FUNCTION_BLOCK FB_DataXMLP3_Old
VAR_INPUT
    	bSave:BOOL;
	    bRead:BOOL;

END_VAR
VAR_OUTPUT
    	bSaveParDone      :BOOL;
	    bReadParDone     :BOOL;
		bError                     :BOOL;		
END_VAR

VAR


	iDataSetp: INT;
	TON10:Tc2_Standard.TON;
	I1: INT;
	rt100:Tc2_Standard.R_TRIG;
	rt101:Tc2_Standard.R_TRIG;
	bExecute1: BOOL;
	bExecute2: BOOL;


	bSaveTemp: BOOL;
	bReadTemp: BOOL;

 fbXmlSrvWrite         : FB_XmlSrvWrite;
// fbXmlSrvWrite         : FB_SrvWrite;
   bExecuteW1             : BOOL;
   sFilePathPar_W       : T_MaxString ;

 
fbXmlSrvRead   : FB_XmlSrvRead;
//fbXmlSrvRead   : FB_SrvRead;
   bExecuteR          : BOOL;
   sFilePathPar_R      : T_MaxString ;
   sXPathR             : T_MaxString;
	AA: INT;
	BB: INT;












	handleTemp: UDINT;
END_VAR


M_WriteOrRead();

ACTION M_WriteOrRead:
bError := fbXmlSrvWrite.bError OR   fbXmlSrvRead.bError;

rt100(CLK:=bSave , Q=> );//保存参数
rt101(CLK:=bRead , Q=> );//读取参数

IF rt100.Q THEN  //保存参数
	iDataSetp:=100;
	TON10.IN:=FALSE;
	I1:=1;
	bExecute1:=FALSE;
	bExecute2:=FALSE;
	bSave:=FALSE;
	bRead:=FALSE;
    bSaveTemp:=TRUE;
	bReadTemp:=FALSE;
	bSaveParDone:=FALSE;
END_IF

IF rt101.Q THEN  //读取参数
	iDataSetp:=100;
	TON10.IN:=FALSE;
	I1:=1;
	bExecute1:=FALSE;
	bExecute2:=FALSE;	
	bSave:=FALSE;
	bRead:=FALSE;
    bReadTemp:=TRUE;
    bSaveTemp:=FALSE;
    bReadParDone:=FALSE;
END_IF

TON10(IN:= , PT:=T#200MS , Q=> , ET=> );

CASE  iDataSetp OF 
	
 100:
				CASE I1 OF 
				  1://轴参数
					sFilePathPar_W  := 'C:\P3XML\P3arrAxisParV2.xml';
					fbXmlSrvWrite.pSymAddr:=ADR(arrAxisParV2);
					fbXmlSrvWrite.cbSymSize:=SIZEOF(arrAxisParV2);   

					sFilePathPar_R  :=  'C:\P3XML\P3arrAxisParV2.xml';
					fbXmlSrvRead.pSymAddr:=ADR(arrAxisParV2);
					fbXmlSrvRead.cbSymSize:=SIZEOF(arrAxisParV2);   
     
				  2://arrTempPar
		  		    sFilePathPar_W  := 'C:\P3XML\P3arrTempPar.xml';
					fbXmlSrvWrite.pSymAddr:=ADR(arrTempPar);
					fbXmlSrvWrite.cbSymSize:=SIZEOF(arrTempPar);     

					sFilePathPar_R  := 'C:\P3XML\P3arrTempPar.xml';
					fbXmlSrvRead.pSymAddr:=ADR(arrTempPar);
					fbXmlSrvRead.cbSymSize:=SIZEOF(arrTempPar);   

				  3://P3par
		  		     sFilePathPar_W  := 'C:\P3XML\P3par.xml';
					fbXmlSrvWrite.pSymAddr:=ADR(P3par);
					fbXmlSrvWrite.cbSymSize:=SIZEOF(P3par);     

					sFilePathPar_R  := 'C:\P3XML\P3par.xml';
					fbXmlSrvRead.pSymAddr:=ADR(P3par);
					fbXmlSrvRead.cbSymSize:=SIZEOF(P3par);   
					
			     4://P3par
		  		     sFilePathPar_W  := 'C:\P3XML\P3User2_Par.xml';
					fbXmlSrvWrite.pSymAddr:=ADR(P3User2_Par);
					fbXmlSrvWrite.cbSymSize:=SIZEOF(P3User2_Par);     

					sFilePathPar_R  := 'C:\P3XML\P3User2_Par.xml';
					fbXmlSrvRead.pSymAddr:=ADR(P3User2_Par);
					fbXmlSrvRead.cbSymSize:=SIZEOF(P3User2_Par);   				
			
				END_CASE
        IF  bSaveTemp THEN
              handleTemp:=fbXmlSrvWrite.handle;
   	          iDataSetp:=200;
       END_IF
        IF  bReadTemp THEN
              handleTemp:=fbXmlSrvRead.handle;
   	          iDataSetp:=300;
       END_IF

	   
	200:	//保存数据
		bExecute1:=TRUE;
        iDataSetp:=210;
	210:	
       IF  NOT fbXmlSrvWrite.bError  AND NOT fbXmlSrvWrite.bBusy AND handleTemp<>fbXmlSrvWrite.handle  THEN
             iDataSetp:=500;
      END_IF
	  
	300:	//读取参数
		bExecute2:=TRUE;
        iDataSetp:=310;
	310:	
       IF  NOT fbXmlSrvRead.bError  AND NOT fbXmlSrvRead.bBusy AND handleTemp<>fbXmlSrvRead.handle  THEN
             iDataSetp:=500;
      END_IF


	500://继续写下个文件
	  IF I1>=1 AND I1<4 THEN
		 I1:=I1+1; 
		 iDataSetp:=100; 
		 bExecute1:=FALSE; 
		 bExecute2:=FALSE; 
	  ELSIF I1>=4 THEN
          IF  bSaveTemp THEN
               bSaveParDone:=TRUE;
         END_IF

          IF  bReadTemp THEN
               bReadParDone:=TRUE;
         END_IF

		  bReadTemp:=FALSE;
          bSaveTemp:=FALSE;

	   	 iDataSetp:=666;   
	  END_IF
END_CASE


AA:=BB;

fbXmlSrvWrite(
   nMode           := XMLSRV_ADDMISSING,
   pSymAddr        :=,//ADR(Value1)
   cbSymSize       := ,//SIZEOF(Value1)
   sFilePath       := sFilePathPar_W,
   sXPath	       := '/dataentry/value',
   bExecute        := bExecute1
);


fbXmlSrvRead(
   pSymAddr       := ,
   cbSymSize      := ,
   sFilePath      := sFilePathPar_R,
   sXPath	         := '/dataentry/value',
   bExecute       := bExecute2
);
END_ACTION

END_FUNCTION_BLOCK

(* stored: Version 1.1.0.1, ProductVersion 3.1.4024.12
   POU FB_DataXMLP3_Old: Id {cc3728ce-ce44-4370-a4e5-7b83fd71ae87}, SpecialFunc None
   Action M_WriteOrRead: Id {55042fcf-47ae-4705-b531-123741cf6044} *)
